FUNCTION_BLOCK EverestMC implements I_Motor
VAR_INPUT
	//
END_VAR
VAR_OUTPUT
END_VAR
VAR
	Axis: AXIS_REF;
	Enabled: BOOL := FALSE;
	Override: LREAL:=100;
	MotorError AT%I*	:WORD;
	MotorErrorSent : WORD;
	AxisErrorSent:UDINT;
	NCError : WORD;
	fbMessage : FB_TcMessage;
	EnableEventSent:BOOL:= TRUE;
	HomeEventSent:BOOL:=TRUE;
	MovementFinishedEventSent:BOOL;
    fbAxisMoveAbsolute: MC_MoveAbsolute;	
	fbMcHome: MC_Home;
	fbAxisPower: MC_Power;
	fbReset: MC_Reset;
	fbMoveRel : MC_MoveRelative;
	
END_VAR

Axis.ReadStatus();

IF NOT (MotorError = MotorErrorSent) THEN// Creates Event 
	MotorErrorSent:= MotorError;
	fbMessage.CreateEx(TC_Events.LinearMotor.IDXmotorError,0);
	fbMessage.ipArguments.Clear().AddDWord(MotorError);
	fbMessage.Send(0);
END_IF

IF NOT (Axis.NcToPlc.ErrorCode = AxisErrorSent) THEN// Creates Event 
	AxisErrorSent:= Axis.NcToPlc.ErrorCode;
	fbMessage.CreateEx(TC_Events.LinearMotor.AxisError,0);
	fbMessage.ipArguments.Clear().AddDWord(Axis.NcToPlc.ErrorCode);
	fbMessage.Send(0);
END_IF

METHOD Enable : BOOL
VAR_INPUT
	EnableMotor :BOOL;
END_VAR
	fbAxisPower( // use in idx class
    Axis:= Axis,
    Enable:= EnableMotor,
    Enable_Positive:= EnableMotor,
    Enable_Negative:= EnableMotor,
    Override:= Override,
	Status=>Enable,
	Error=>
);

IF EnableMotor = EnableEventSent THEN	
	EnableEventSent := NOT EnableEventSent;
IF EnableMotor THEN
	fbMessage.CreateEx(TC_Events.LinearMotor.Motor_enabled,0);
ELSE
	fbMessage.CreateEx(TC_Events.LinearMotor.Motor_disabled,0);
END_IF
//fbMessage.Send(0);
END_IF
END_METHOD

METHOD Estop : BOOL
VAR_INPUT
END_VAR
END_METHOD

METHOD PUBLIC Home : BOOL
VAR_IN_OUT
	Execute:BOOL;
END_VAR
VAR
	HomingDone:BOOL;
	HomingError:BOOL;
	HomingErrorID:UDINT;
END_VAR
// try changing limits to no error mode then home 


	fbMcHome(
	Axis:=Axis,
	Execute:=Execute,
	//Position:=510,
	HomingMode:=MC_DefaultHoming,
	Busy=>Home,
	Done=>HomingDone,
	Error=> HomingError,
	ErrorID=> HomingErrorID
);
	
IF Execute THEN
	HomeEventSent:= FALSE;
	fbMessage.CreateEx(TC_Events.LinearMotor.Homing,0);
	//fbMessage.Send(0);
	Execute:= FALSE;	
END_IF
IF HomingDone THEN
	fbMessage.CreateEx(TC_Events.LinearMotor.HomingComplete,0);
	//fbMessage.Send(0);
END_IF

IF HomingError THEN
	fbMessage.CreateEx(TC_Events.LinearMotor.HomingFailed,0);
	fbMessage.ipArguments.Clear().AddDWord(HomingErrorID);
	//fbMessage.Send(0);
END_IF
END_METHOD

METHOD PUBLIC Homed : BOOL
VAR_INPUT
END_VAR
Homed:=Axis.NcToPlc.StateDWord.1;
END_METHOD

METHOD MoveRelative : BOOL
VAR_INPUT
	Distance: LREAL;
	Velocity: LREAL;	
END_VAR
VAR_IN_OUT
	Execute: BOOL;
END_VAR
	fbMoveRel( // in idx class 
    Axis:= Axis,
    Execute:= Execute,
    Distance:= Distance,
    Velocity:= Velocity,);
	
		IF Execute THEN
	fbMessage.CreateEx(TC_Events.LinearMotor.RelativeMove,0);
	fbMessage.ipArguments.Clear();
	fbMessage.ipArguments.AddLReal(Distance);
	fbMessage.ipArguments.AddLReal(Velocity);
	//fbMessage.Send(0);
	Execute := FALSE;
END_IF

IF fbMoveRel.Done  THEN
	fbMessage.CreateEx(TC_Events.LinearMotor.MoveComplete,0);
	//fbMessage.Send(0);
	
END_IF
END_METHOD

METHOD PUBLIC MoveTo : BOOL
VAR_INPUT
	Position: LREAL;
	Velocity: LREAL;	
END_VAR

VAR_OUTPUT
	State:e_MCState;
	Target : LREAL;
END_VAR

VAR_IN_OUT
		Execute: BOOL;
END_VAR
 	fbAxisMoveAbsolute( // in idx class 
    Axis:= Axis,
    Execute:= Execute,
    Position:= Position,
    Velocity:= Velocity,);
	
	IF Execute THEN
	fbMessage.CreateEx(TC_Events.LinearMotor.MotorMove,0);
	fbMessage.ipArguments.Clear();
	fbMessage.ipArguments.AddLReal(Position);
	fbMessage.ipArguments.AddLReal(Velocity);
	//fbMessage.Send(0);
	Execute := FALSE;

END_IF

IF fbAxisMoveAbsolute.Done  THEN
	fbMessage.CreateEx(TC_Events.LinearMotor.MoveComplete,0);
	//fbMessage.Send(0);

	
END_IF
END_METHOD

METHOD Position : LREAL
VAR_INPUT
END_VAR
Position:= Axis.NcToPlc.ActPos;
END_METHOD

METHOD Reset : BOOL
VAR_IN_OUT
	ResetAxis:BOOL;
END_VAR
fbReset(
Axis:=Axis,
Execute:=ResetAxis,
Done =>Reset);

IF resetAxis THEN
//IDXControlByte1 := 16#80;// restop linear Motor
//MotorResetBit := 16#80;
fbMessage.CreateEx(TC_Events.LinearMotor.AxisReset,0);
//fbMessage.send(0);
resetAxis := FALSE;
END_IF
END_METHOD

METHOD PUBLIC Status : ST_AxisStatus
VAR_INPUT
END_VAR
Status := Axis.Status;
END_METHOD

END_FUNCTION_BLOCK

(* stored: Version 1.1.0.1, ProductVersion 3.1.4024.12
   POU EverestMC: Id {a3e9c92e-64fa-4e46-a3aa-714fb5bbcbd7}, SpecialFunc None
   Method Enable: Id {7ad8bb3b-6b12-422c-9078-6bc6263f2138}
   Method Estop: Id {035e129b-fd86-43a8-8068-42279faecb42}
   Method Home: Id {ff6a7707-04a2-4925-89cf-1f17c30273a4}
   Method Homed: Id {c997b53f-68dd-42d9-ade9-e7a024632056}
   Method MoveRelative: Id {493795df-a0ca-47e4-90a1-99a456e23940}
   Method MoveTo: Id {4cd2771e-ffe3-4a96-9535-c052480de063}
   Method Position: Id {93992187-0b52-47e0-918d-28c0417601fd}
   Method Reset: Id {9478a509-1996-4742-b1cb-06b31e7be6ec}
   Method Status: Id {c8dd27f2-b4b5-44a3-97d2-a6ab733a23e6} *)
